{attribute 'GeneratedUsingTerminal: ELM9410-0000-0016'}
{attribute addProperty BoxType "ELM9410-0000-0016"}
{attribute addProperty Id "EtcSlaveTerminalBaseMMS_Device_InputsAT %I*MMS_Device_Inputs_7D6F87344MMS_Acceleration_StatusAT %I*MMS_Acceleration_Status_117690999MMS_Acceleration_X_AxisAT %I*MMS_Acceleration_X_Axis_80E77D6A2MMS_Acceleration_Y_AxisAT %I*MMS_Acceleration_Y_Axis_80E77D6A2MMS_Acceleration_Z_AxisAT %I*MMS_Acceleration_Z_Axis_80E77D6A2MMS_Acceleration_TimestampAT %I*MMS_Acceleration_Timestamp_8B9FE1A28MMS_Voltage_Us_In_InputsAT %I*MMS_Voltage_Us_In_Inputs_60D55C7211MMS_Voltage_Up_In_InputsAT %I*MMS_Voltage_Up_In_Inputs_60D55C7211MMS_Voltage_Up_Out_InputsAT %I*MMS_Voltage_Up_Out_Inputs_60D55C7211MMS_Device_OutputsAT %Q*MMS_Device_Outputs_E6E6F9D11WcStateAT %I*WcState_9091E0EB2InfoDataAT %I*InfoData_BEF6B88E18"}
{attribute addProperty CRC "324325699"}
{attribute addProperty Size "81"}
TYPE ELM9410_1354D143 EXTENDS EtcSlaveTerminalBase :
STRUCT
	{attribute addProperty Name "MMS_Device_Inputs"}
	MMS_Device_Inputs : MMS_Device_Inputs_7D6F8734;
	{attribute addProperty Name "MMS_Acceleration_Status"}
	MMS_Acceleration_Status : MMS_Acceleration_Status_11769099;
	{attribute addProperty Name "MMS_Acceleration_X_Axis"}
	MMS_Acceleration_X_Axis : MMS_Acceleration_X_Axis_80E77D6A;
	{attribute addProperty Name "MMS_Acceleration_Y_Axis"}
	MMS_Acceleration_Y_Axis : MMS_Acceleration_Y_Axis_80E77D6A;
	{attribute addProperty Name "MMS_Acceleration_Z_Axis"}
	MMS_Acceleration_Z_Axis : MMS_Acceleration_Z_Axis_80E77D6A;
	{attribute addProperty Name "MMS_Acceleration_Timestamp"}
	MMS_Acceleration_Timestamp : MMS_Acceleration_Timestamp_8B9FE1A2;
	{attribute addProperty Name "MMS_Voltage_Us_In_Inputs"}
	MMS_Voltage_Us_In_Inputs : MMS_Voltage_Us_In_Inputs_60D55C72;
	{attribute addProperty Name "MMS_Voltage_Up_In_Inputs"}
	MMS_Voltage_Up_In_Inputs : MMS_Voltage_Up_In_Inputs_60D55C72;
	{attribute addProperty Name "MMS_Voltage_Up_Out_Inputs"}
	MMS_Voltage_Up_Out_Inputs : MMS_Voltage_Up_Out_Inputs_60D55C72;
	{attribute addProperty Name "MMS_Device_Outputs"}
	MMS_Device_Outputs : MMS_Device_Outputs_E6E6F9D1;
	{attribute addProperty Name "WcState"}
	WcState : WcState_9091E0EB;
	{attribute addProperty Name "InfoData"}
	InfoData : InfoData_BEF6B88E;
END_STRUCT
END_TYPE

(* stored: Version 1.2.0.0, ProductVersion 3.1.4024.9
   DUT ELM9410_1354D143: Id {24268359-7d48-44c6-b351-d2a9b59a0670} *)
